// TIA Portal V17 export
// export: Created 2023-02-26T22:59:50.1784682Z, ExportSetting WithDefaults, DisplayName Totally Integrated Automation Portal, DisplayVersion V17, DisplayName TIA Portal Openness, DisplayVersion V17, DisplayName TIA Portal Version Control Interface, DisplayVersion V17, DisplayName TIA Portal Test Suite Advanced, DisplayVersion V17, DisplayName STEP 7 Professional, DisplayVersion V17, DisplayName SIMATIC Energy Suite, DisplayVersion V17, DisplayName STEP 7 Safety, DisplayVersion V17, DisplayName WinCC Professional, DisplayVersion V17
DATA_BLOCK "LOG_ConveyorWorkTime"   // DB47
{ S7_Optimized_Access := 'TRUE' }
VERSION : 0.1
// stored: AutoNumber true, IsOnlyStoredInLoadMemory false, IsRetainMemResEnabled false, IsWriteProtectedInAS false, MemoryReserve 20
   VAR RETAIN
      T1 { S7_SetPoint := 'True'} : "stt_TimeWork";
      T2 { S7_SetPoint := 'True'} : "stt_TimeWork";
      T3 { S7_SetPoint := 'True'} : "stt_TimeWork";
   END_VAR
   VAR
      T4 { S7_SetPoint := 'True'} : "stt_TimeWork";
      W { S7_SetPoint := 'True'} : "stt_TimeWork";
      O { S7_SetPoint := 'True'} : "stt_TimeWork";
   END_VAR
BEGIN
END_DATA_BLOCK
